FUNCTION_BLOCK E_T_FF_Dual (* Toggle flip flop *)
  (* Standard: 61499-1 Annex A; Description: Copyright (c) 2017 fortiss GmbH This program and the accompanying materials are made available under the terms of the Eclipse Public License 2.0 which is available at https://www.eclipse.org/legal/epl-2.0/ SPDX-License-Identifier: EPL-2.0 *)
  (* Version 1.0, 2017-09-22, Alois Zoitl, fortiss GmbH, initial API and implementation and/or initial documentation *)
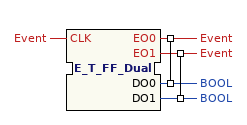
  EVENT_INPUT
    CLK; (* Clock for triggering a output toggle *)
  END_EVENT
  EVENT_OUTPUT
    EO0 WITH DO0; (* inform of toggled output 0 *)
    EO1 WITH DO1; (* inform of toggled output 1 *)
  END_EVENT
  VAR_OUTPUT
    DO0 : BOOL; (* value of flip flop 0 *)
    DO1 : BOOL; (* value of flip flop 1 *)
  END_VAR
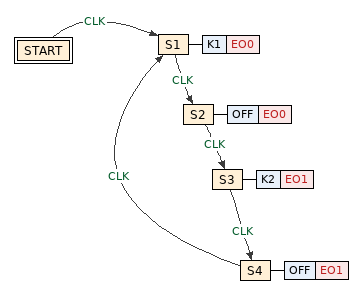
  EC_STATES
    START; (* Initial State *)
    S1 : K1 -> EO0; (* Initialization *)
    S2 : OFF -> EO0;
    S3 : K2 -> EO1;
    S4 : OFF -> EO1;
  END_STATES
  EC_TRANSITIONS
    START TO S1 := CLK;
    S1 TO S2 := CLK;
    S2 TO S3 := CLK;
    S3 TO S4 := CLK;
    S4 TO S1 := CLK;
  END_TRANSITIONS
  ALGORITHM OFF IN ST: (* new algorithm *)
DO0 := FALSE; DO1 := FALSE;
  END_ALGORITHM
  ALGORITHM K1 IN ST: (* new algorithm *)
DO0 := TRUE; DO1 := FALSE;
  END_ALGORITHM
  ALGORITHM K2 IN ST: (* new algorithm *)
DO0 := FALSE; DO1 := TRUE;
  END_ALGORITHM
END_FUNCTION_BLOCK
